(* Logix 5000 project; controller cal1632 1756-L62 rev 16.20; software revision 16.05; part 37 of 61 *)
(* tags used below, declared in another part *)
   FAULT : BOOL;
   HMI : BOOL;
   p01r09_pb_global_reset : BOOL;
   p23_ao_selected_speed : REAL;
   p23_ao_servo_ds_jog_vel_cmd : REAL;
   p23_ao_servo_ds_position_cmd : REAL;
   p23_ao_servo_ds_velocity_cmd : REAL;
   p23_ao_servo_ds_zero_offset : REAL;
   p23_ao_servo_os_jog_vel_cmd : REAL;
   p23_ao_servo_os_position_cmd : REAL;
   p23_ao_servo_os_velocity_cmd : REAL;
   p23_ao_servo_os_zero_offset : REAL;
   p23_ao_supply_selected_speed : REAL;
   p23_cpr_gear_ratio : REAL;
   p23_cpr_roll_diameter_ft : REAL;
   p23_cpr_speed_to_vfd : SYS_SPEED_TO_VFD;
   p23_di_impreg_tank_up : BOOL;
   p23_di_metering_roll : acs800_di_normal;
   p23_di_servo_ds : servo_di;
   p23_di_servo_os : servo_di;
   p23_di_supply : acs800_di_normal;
   p23_di_tank_level_high : BOOL;
   p23_di_tank_level_low : BOOL;
   p23_di_though_level_low : BOOL;
   p23_dint_to_hmi : DINT[32];
   p23_do_enable_impreg_exhaust_fan : BOOL;
   p23_do_enable_impreg_supply_fan : BOOL;
   p23_do_impreg : acs800_do_normal;
   p23_do_impreg_nip_close : BOOL;
   p23_do_servo_ds : servo_do;
   p23_do_servo_os : servo_do;
   p23_do_Spring : acs800_do_normal;
   p23_do_supply : acs800_do_normal;
   p23_servo_ds_error : SYS_ENC_WITH_ZERO_BIT;
   p23_servo_ds_warning : SYS_ENC_WITH_ZERO_BIT;
   p23_servo_os_error : SYS_ENC_WITH_ZERO_BIT;
   p23_servo_os_warning : SYS_ENC_WITH_ZERO_BIT;
   p23_spring_gear_ratio : REAL;
   p23_spring_roll_diameter_ft : REAL;
   p23_spring_speed_to_vfd : SYS_SPEED_TO_VFD;
   p23r04 : routine;
   p23r04_timer_fault : TIMER[4];
   p23r04_timer_warning : TIMER[4];
   p23r05 : routine;
   p23r05_supply_status : DINT;
   p23r05_timer_fault : TIMER[4];
   p23r05_timer_warning : TIMER[4];
   p23r11_servo_not_ready : BOOL;
   p23r11_servo_status_ab : BOOL;
   p23r11_servo_status_af : BOOL;
   p23r11_servo_status_bb : BOOL;
   p23r12_servo_not_ready : BOOL;
   p23r12_servo_status_ab : BOOL;
   p23r12_servo_status_af : BOOL;
   p23r12_servo_status_bb : BOOL;
   p23r13 : routine;
   p23r13_vfd_stopped : BOOL;
   p23r15_pid_tension_control : BOOL;
   p23r17_adjusted_speed : REAL;
   p32r13_request_auto_stop : BOOL;
(* P23_Impreg, continued *)

ROUTINE R04_Outputs   (* ladder *)
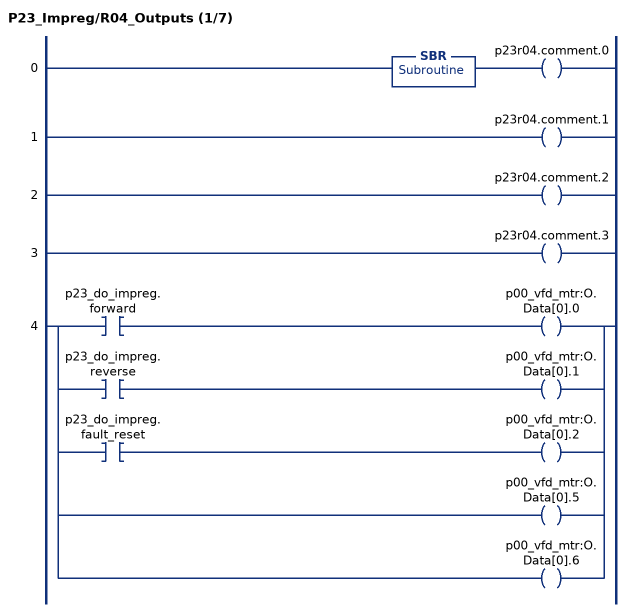
   0: SBR()OTE(p23r04.comment.0);
   1: OTE(p23r04.comment.1);
   2: OTE(p23r04.comment.2);
   3: OTE(p23r04.comment.3);
   4: [XIC(p23_do_impreg.forward) OTE(p00_vfd_mtr:O.Data[0].0) ,XIC(p23_do_impreg.reverse) OTE(p00_vfd_mtr:O.Data[0].1) ,XIC(p23_do_impreg.fault_reset) OTE(p00_vfd_mtr:O.Data[0].2) ,OTE(p00_vfd_mtr:O.Data[0].5) ,OTE(p00_vfd_mtr:O.Data[0].6) ];
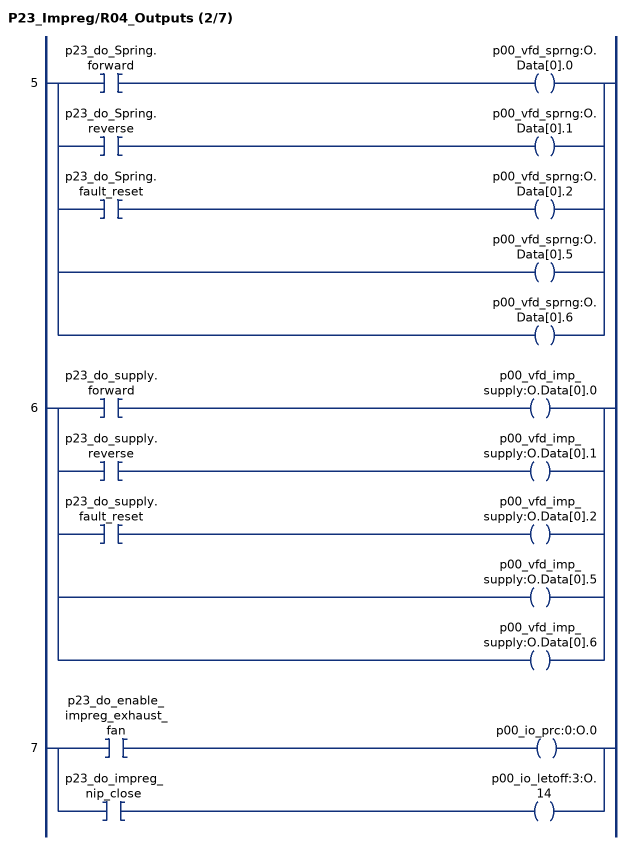
   5: [XIC(p23_do_Spring.forward) OTE(p00_vfd_sprng:O.Data[0].0) ,XIC(p23_do_Spring.reverse) OTE(p00_vfd_sprng:O.Data[0].1) ,XIC(p23_do_Spring.fault_reset) OTE(p00_vfd_sprng:O.Data[0].2) ,OTE(p00_vfd_sprng:O.Data[0].5) ,OTE(p00_vfd_sprng:O.Data[0].6) ];
   6: [XIC(p23_do_supply.forward) OTE(p00_vfd_imp_supply:O.Data[0].0) ,XIC(p23_do_supply.reverse) OTE(p00_vfd_imp_supply:O.Data[0].1) ,XIC(p23_do_supply.fault_reset) OTE(p00_vfd_imp_supply:O.Data[0].2) ,OTE(p00_vfd_imp_supply:O.Data[0].5) ,OTE(p00_vfd_imp_supply:O.Data[0].6) ];
   7: [XIC(p23_do_enable_impreg_exhaust_fan) OTE(p00_io_prc:0:O.0) ,XIC(p23_do_impreg_nip_close) OTE(p00_io_letoff:3:O.14) ];
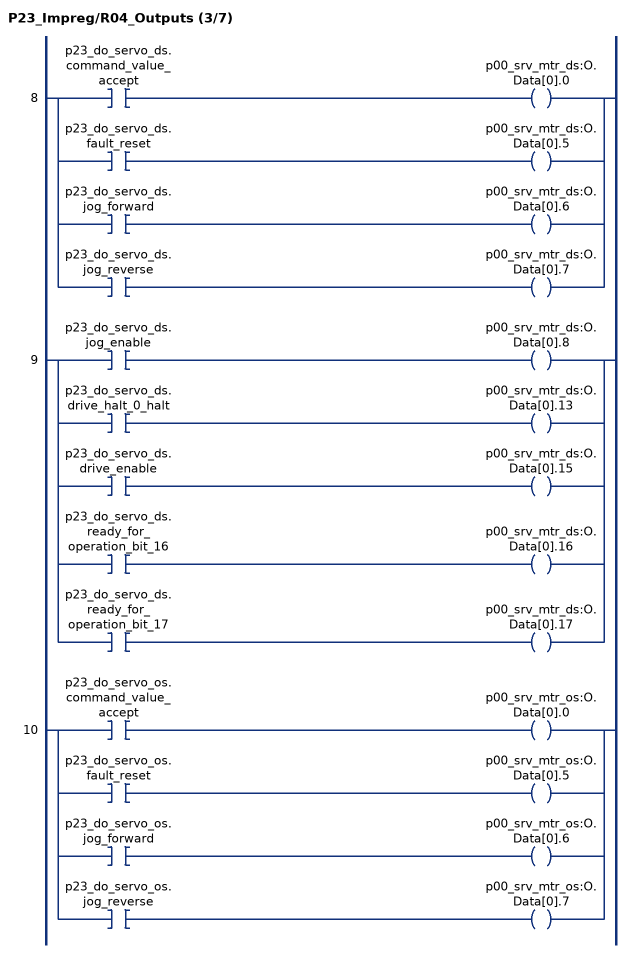
   8: [XIC(p23_do_servo_ds.command_value_accept) OTE(p00_srv_mtr_ds:O.Data[0].0) ,XIC(p23_do_servo_ds.fault_reset) OTE(p00_srv_mtr_ds:O.Data[0].5) ,XIC(p23_do_servo_ds.jog_forward) OTE(p00_srv_mtr_ds:O.Data[0].6) ,XIC(p23_do_servo_ds.jog_reverse) OTE(p00_srv_mtr_ds:O.Data[0].7) ];
   9: [XIC(p23_do_servo_ds.jog_enable) OTE(p00_srv_mtr_ds:O.Data[0].8) ,XIC(p23_do_servo_ds.drive_halt_0_halt) OTE(p00_srv_mtr_ds:O.Data[0].13) ,XIC(p23_do_servo_ds.drive_enable) OTE(p00_srv_mtr_ds:O.Data[0].15) ,XIC(p23_do_servo_ds.ready_for_operation_bit_16) OTE(p00_srv_mtr_ds:O.Data[0].16) ,XIC(p23_do_servo_ds.ready_for_operation_bit_17) OTE(p00_srv_mtr_ds:O.Data[0].17) ];
   10: [XIC(p23_do_servo_os.command_value_accept) OTE(p00_srv_mtr_os:O.Data[0].0) ,XIC(p23_do_servo_os.fault_reset) OTE(p00_srv_mtr_os:O.Data[0].5) ,XIC(p23_do_servo_os.jog_forward) OTE(p00_srv_mtr_os:O.Data[0].6) ,XIC(p23_do_servo_os.jog_reverse) OTE(p00_srv_mtr_os:O.Data[0].7) ];
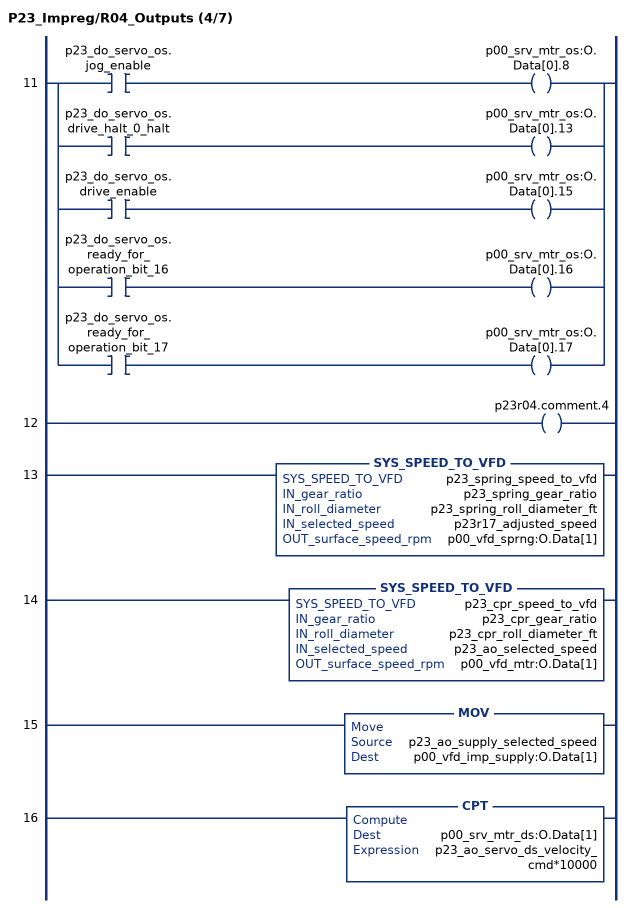
   11: [XIC(p23_do_servo_os.jog_enable) OTE(p00_srv_mtr_os:O.Data[0].8) ,XIC(p23_do_servo_os.drive_halt_0_halt) OTE(p00_srv_mtr_os:O.Data[0].13) ,XIC(p23_do_servo_os.drive_enable) OTE(p00_srv_mtr_os:O.Data[0].15) ,XIC(p23_do_servo_os.ready_for_operation_bit_16) OTE(p00_srv_mtr_os:O.Data[0].16) ,XIC(p23_do_servo_os.ready_for_operation_bit_17) OTE(p00_srv_mtr_os:O.Data[0].17) ];
   12: OTE(p23r04.comment.4);
   13: SYS_SPEED_TO_VFD(p23_spring_speed_to_vfd,p23_spring_gear_ratio,p23_spring_roll_diameter_ft,p23r17_adjusted_speed,p00_vfd_sprng:O.Data[1]);
   14: SYS_SPEED_TO_VFD(p23_cpr_speed_to_vfd,p23_cpr_gear_ratio,p23_cpr_roll_diameter_ft,p23_ao_selected_speed,p00_vfd_mtr:O.Data[1]);
   15: MOV(p23_ao_supply_selected_speed,p00_vfd_imp_supply:O.Data[1]);
   16: CPT(p00_srv_mtr_ds:O.Data[1],p23_ao_servo_ds_velocity_cmd*10000);
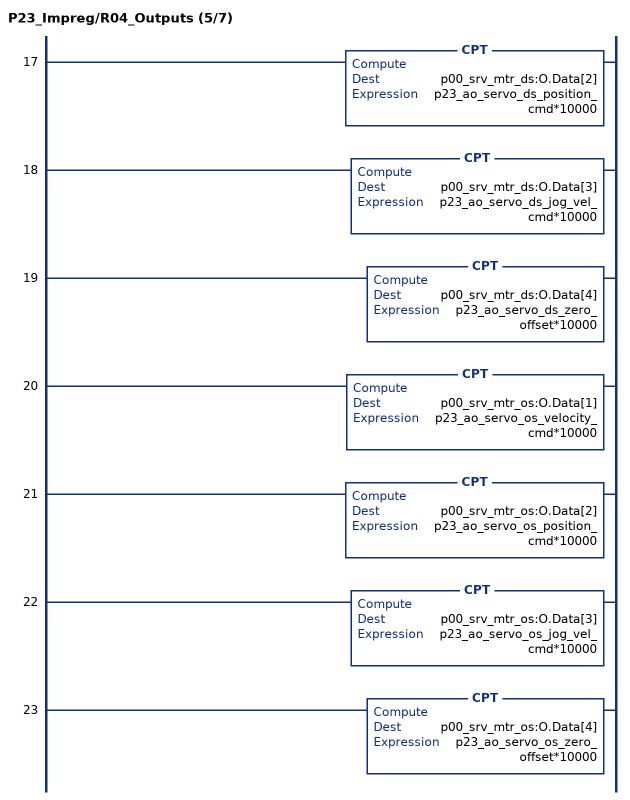
   17: CPT(p00_srv_mtr_ds:O.Data[2],p23_ao_servo_ds_position_cmd*10000);
   18: CPT(p00_srv_mtr_ds:O.Data[3],p23_ao_servo_ds_jog_vel_cmd*10000);
   19: CPT(p00_srv_mtr_ds:O.Data[4],p23_ao_servo_ds_zero_offset*10000);
   20: CPT(p00_srv_mtr_os:O.Data[1],p23_ao_servo_os_velocity_cmd*10000);
   21: CPT(p00_srv_mtr_os:O.Data[2],p23_ao_servo_os_position_cmd*10000);
   22: CPT(p00_srv_mtr_os:O.Data[3],p23_ao_servo_os_jog_vel_cmd*10000);
   23: CPT(p00_srv_mtr_os:O.Data[4],p23_ao_servo_os_zero_offset*10000);
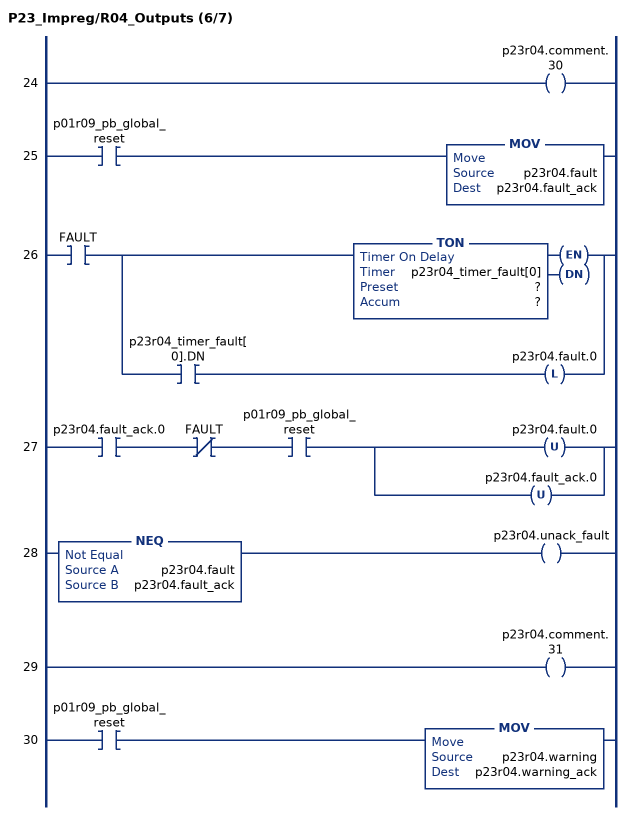
   24: OTE(p23r04.comment.30);
   25: XIC(p01r09_pb_global_reset)MOV(p23r04.fault,p23r04.fault_ack);
   26: XIC(FAULT)[TON(p23r04_timer_fault[0],?,?) ,XIC(p23r04_timer_fault[0].DN) OTL(p23r04.fault.0) ];
   27: XIC(p23r04.fault_ack.0)XIO(FAULT)XIC(p01r09_pb_global_reset)[OTU(p23r04.fault.0) ,OTU(p23r04.fault_ack.0) ];
   28: NEQ(p23r04.fault,p23r04.fault_ack)OTE(p23r04.unack_fault);
   29: OTE(p23r04.comment.31);
   30: XIC(p01r09_pb_global_reset)MOV(p23r04.warning,p23r04.warning_ack);
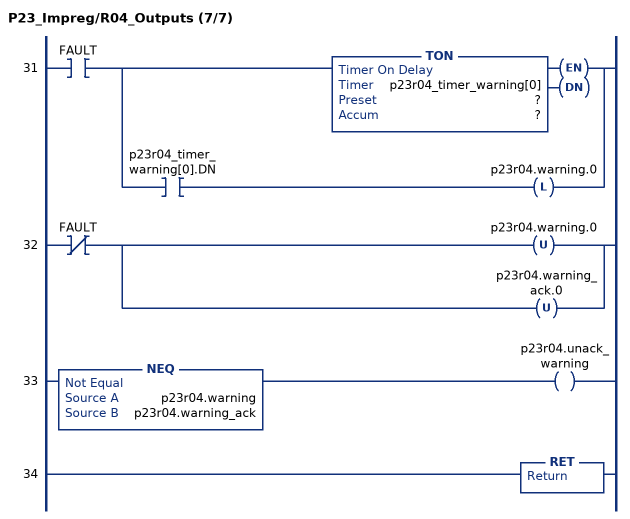
   31: XIC(FAULT)[TON(p23r04_timer_warning[0],?,?) ,XIC(p23r04_timer_warning[0].DN) OTL(p23r04.warning.0) ];
   32: XIO(FAULT)[OTU(p23r04.warning.0) ,OTU(p23r04.warning_ack.0) ];
   33: NEQ(p23r04.warning,p23r04.warning_ack)OTE(p23r04.unack_warning);
   34: RET();
END_ROUTINE

ROUTINE R05_Dint_to_HMI   (* ladder *)
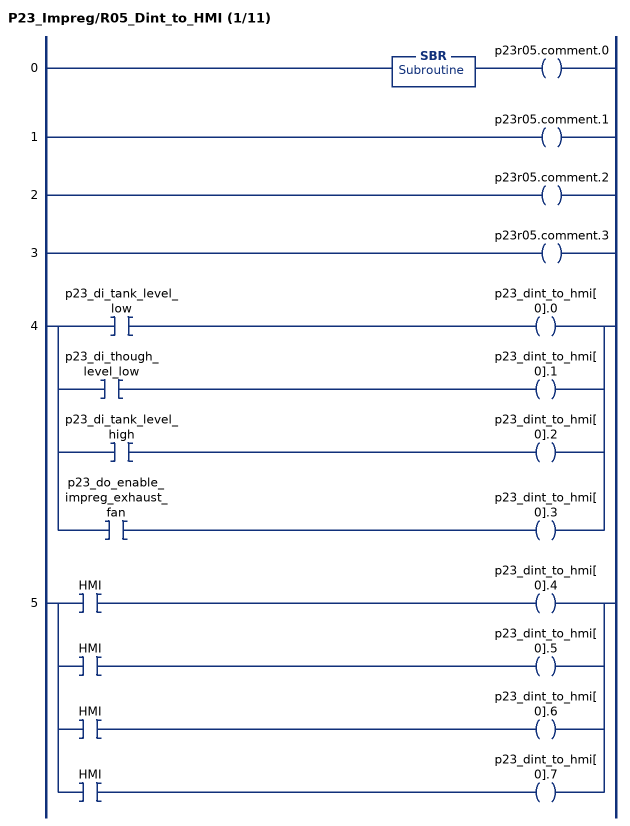
   0: SBR()OTE(p23r05.comment.0);
   1: OTE(p23r05.comment.1);
   2: OTE(p23r05.comment.2);
   3: OTE(p23r05.comment.3);
   4: [XIC(p23_di_tank_level_low) OTE(p23_dint_to_hmi[0].0) ,XIC(p23_di_though_level_low) OTE(p23_dint_to_hmi[0].1) ,XIC(p23_di_tank_level_high) OTE(p23_dint_to_hmi[0].2) ,XIC(p23_do_enable_impreg_exhaust_fan) OTE(p23_dint_to_hmi[0].3) ];
   5: [XIC(HMI) OTE(p23_dint_to_hmi[0].4) ,XIC(HMI) OTE(p23_dint_to_hmi[0].5) ,XIC(HMI) OTE(p23_dint_to_hmi[0].6) ,XIC(HMI) OTE(p23_dint_to_hmi[0].7) ];
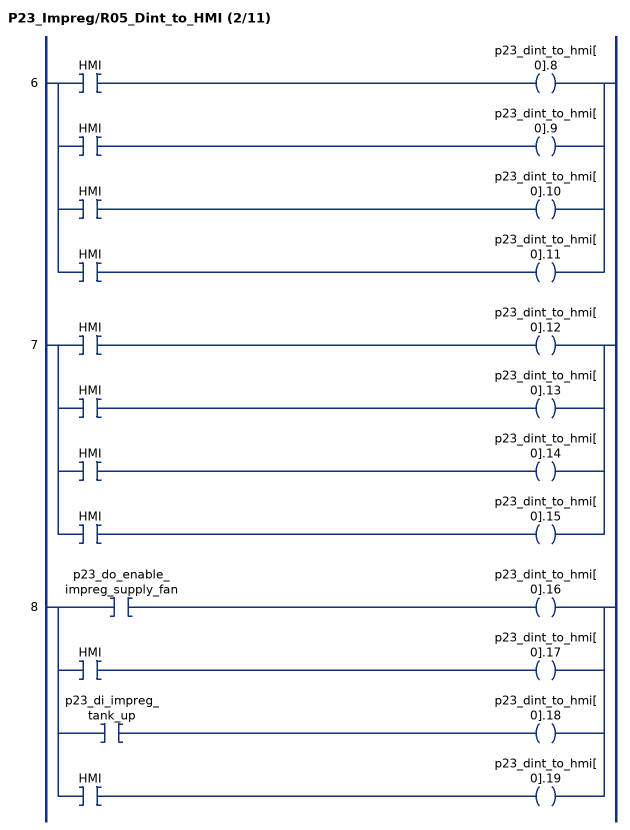
   6: [XIC(HMI) OTE(p23_dint_to_hmi[0].8) ,XIC(HMI) OTE(p23_dint_to_hmi[0].9) ,XIC(HMI) OTE(p23_dint_to_hmi[0].10) ,XIC(HMI) OTE(p23_dint_to_hmi[0].11) ];
   7: [XIC(HMI) OTE(p23_dint_to_hmi[0].12) ,XIC(HMI) OTE(p23_dint_to_hmi[0].13) ,XIC(HMI) OTE(p23_dint_to_hmi[0].14) ,XIC(HMI) OTE(p23_dint_to_hmi[0].15) ];
   8: [XIC(p23_do_enable_impreg_supply_fan) OTE(p23_dint_to_hmi[0].16) ,XIC(HMI) OTE(p23_dint_to_hmi[0].17) ,XIC(p23_di_impreg_tank_up) OTE(p23_dint_to_hmi[0].18) ,XIC(HMI) OTE(p23_dint_to_hmi[0].19) ];
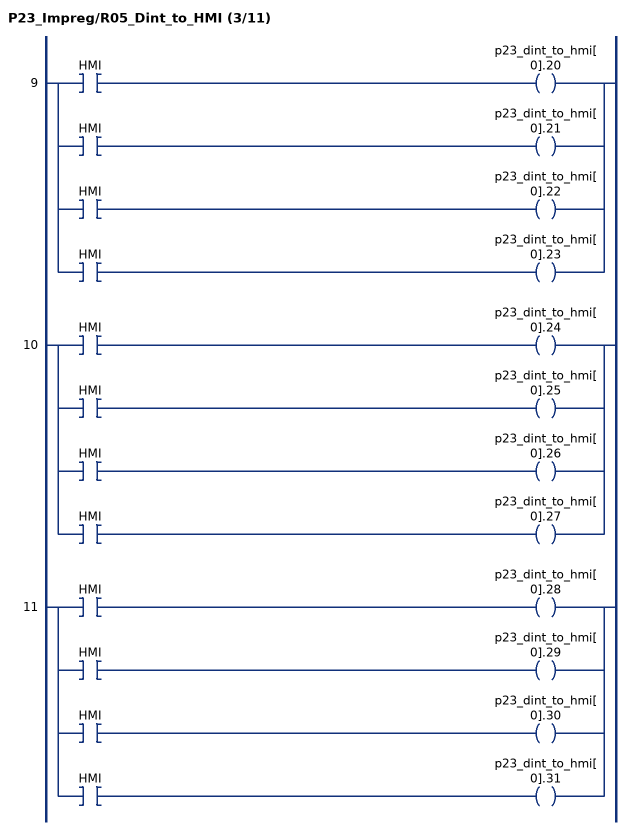
   9: [XIC(HMI) OTE(p23_dint_to_hmi[0].20) ,XIC(HMI) OTE(p23_dint_to_hmi[0].21) ,XIC(HMI) OTE(p23_dint_to_hmi[0].22) ,XIC(HMI) OTE(p23_dint_to_hmi[0].23) ];
   10: [XIC(HMI) OTE(p23_dint_to_hmi[0].24) ,XIC(HMI) OTE(p23_dint_to_hmi[0].25) ,XIC(HMI) OTE(p23_dint_to_hmi[0].26) ,XIC(HMI) OTE(p23_dint_to_hmi[0].27) ];
   11: [XIC(HMI) OTE(p23_dint_to_hmi[0].28) ,XIC(HMI) OTE(p23_dint_to_hmi[0].29) ,XIC(HMI) OTE(p23_dint_to_hmi[0].30) ,XIC(HMI) OTE(p23_dint_to_hmi[0].31) ];
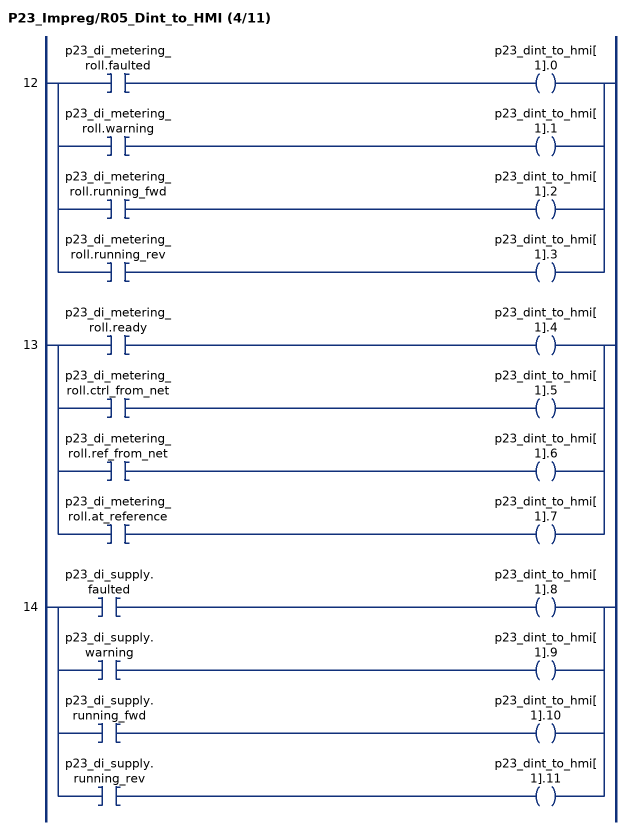
   12: [XIC(p23_di_metering_roll.faulted) OTE(p23_dint_to_hmi[1].0) ,XIC(p23_di_metering_roll.warning) OTE(p23_dint_to_hmi[1].1) ,XIC(p23_di_metering_roll.running_fwd) OTE(p23_dint_to_hmi[1].2) ,XIC(p23_di_metering_roll.running_rev) OTE(p23_dint_to_hmi[1].3) ];
   13: [XIC(p23_di_metering_roll.ready) OTE(p23_dint_to_hmi[1].4) ,XIC(p23_di_metering_roll.ctrl_from_net) OTE(p23_dint_to_hmi[1].5) ,XIC(p23_di_metering_roll.ref_from_net) OTE(p23_dint_to_hmi[1].6) ,XIC(p23_di_metering_roll.at_reference) OTE(p23_dint_to_hmi[1].7) ];
   14: [XIC(p23_di_supply.faulted) OTE(p23_dint_to_hmi[1].8) ,XIC(p23_di_supply.warning) OTE(p23_dint_to_hmi[1].9) ,XIC(p23_di_supply.running_fwd) OTE(p23_dint_to_hmi[1].10) ,XIC(p23_di_supply.running_rev) OTE(p23_dint_to_hmi[1].11) ];
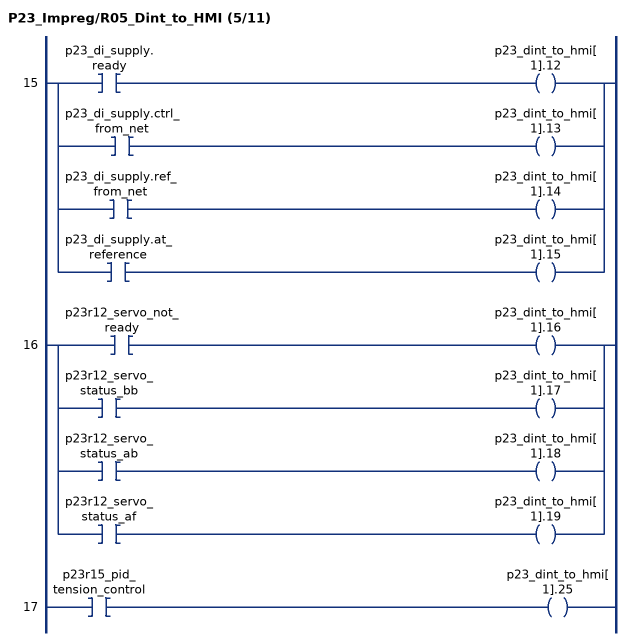
   15: [XIC(p23_di_supply.ready) OTE(p23_dint_to_hmi[1].12) ,XIC(p23_di_supply.ctrl_from_net) OTE(p23_dint_to_hmi[1].13) ,XIC(p23_di_supply.ref_from_net) OTE(p23_dint_to_hmi[1].14) ,XIC(p23_di_supply.at_reference) OTE(p23_dint_to_hmi[1].15) ];
   16: [XIC(p23r12_servo_not_ready) OTE(p23_dint_to_hmi[1].16) ,XIC(p23r12_servo_status_bb) OTE(p23_dint_to_hmi[1].17) ,XIC(p23r12_servo_status_ab) OTE(p23_dint_to_hmi[1].18) ,XIC(p23r12_servo_status_af) OTE(p23_dint_to_hmi[1].19) ];
   17: XIC(p23r15_pid_tension_control)OTE(p23_dint_to_hmi[1].25);
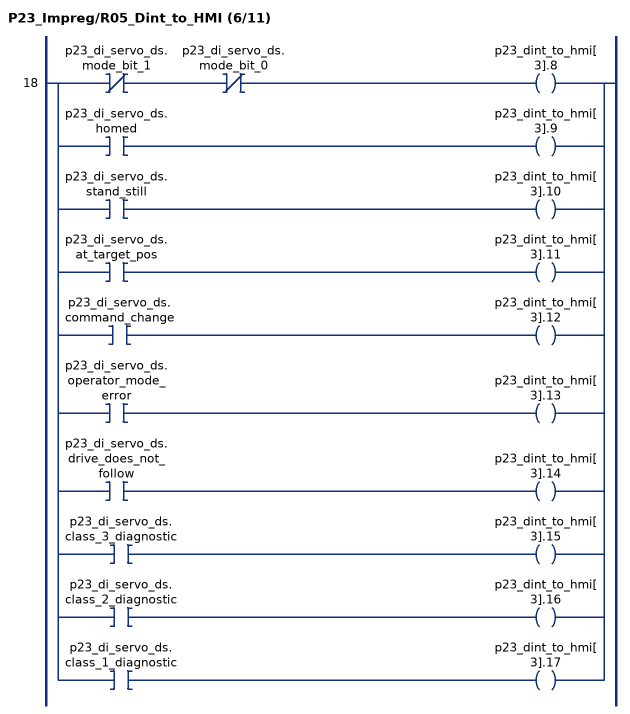
   18: [XIO(p23_di_servo_ds.mode_bit_1) XIO(p23_di_servo_ds.mode_bit_0) OTE(p23_dint_to_hmi[3].8) ,XIC(p23_di_servo_ds.homed) OTE(p23_dint_to_hmi[3].9) ,XIC(p23_di_servo_ds.stand_still) OTE(p23_dint_to_hmi[3].10) ,XIC(p23_di_servo_ds.at_target_pos) OTE(p23_dint_to_hmi[3].11) ,XIC(p23_di_servo_ds.command_change) OTE(p23_dint_to_hmi[3].12) ,XIC(p23_di_servo_ds.operator_mode_error) OTE(p23_dint_to_hmi[3].13) ,XIC(p23_di_servo_ds.drive_does_not_follow) OTE(p23_dint_to_hmi[3].14) ,XIC(p23_di_servo_ds.class_3_diagnostic) OTE(p23_dint_to_hmi[3].15) ,XIC(p23_di_servo_ds.class_2_diagnostic) OTE(p23_dint_to_hmi[3].16) ,XIC(p23_di_servo_ds.class_1_diagnostic) OTE(p23_dint_to_hmi[3].17) ];
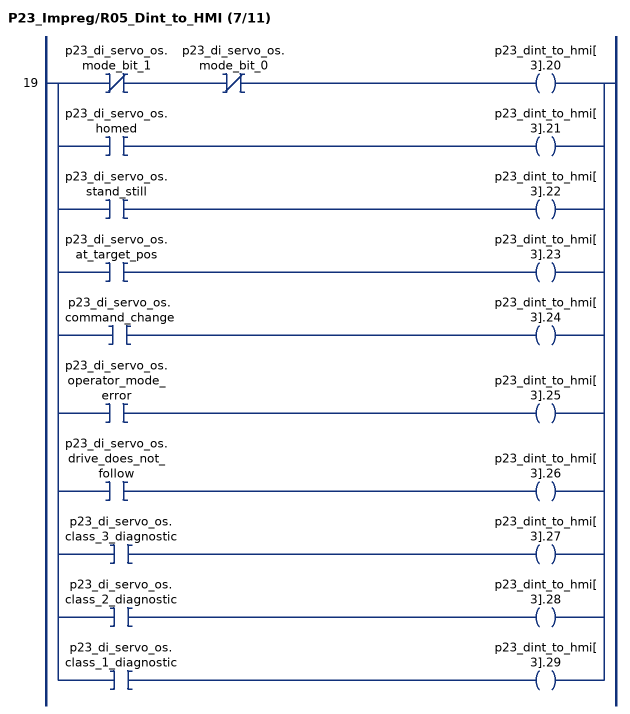
   19: [XIO(p23_di_servo_os.mode_bit_1) XIO(p23_di_servo_os.mode_bit_0) OTE(p23_dint_to_hmi[3].20) ,XIC(p23_di_servo_os.homed) OTE(p23_dint_to_hmi[3].21) ,XIC(p23_di_servo_os.stand_still) OTE(p23_dint_to_hmi[3].22) ,XIC(p23_di_servo_os.at_target_pos) OTE(p23_dint_to_hmi[3].23) ,XIC(p23_di_servo_os.command_change) OTE(p23_dint_to_hmi[3].24) ,XIC(p23_di_servo_os.operator_mode_error) OTE(p23_dint_to_hmi[3].25) ,XIC(p23_di_servo_os.drive_does_not_follow) OTE(p23_dint_to_hmi[3].26) ,XIC(p23_di_servo_os.class_3_diagnostic) OTE(p23_dint_to_hmi[3].27) ,XIC(p23_di_servo_os.class_2_diagnostic) OTE(p23_dint_to_hmi[3].28) ,XIC(p23_di_servo_os.class_1_diagnostic) OTE(p23_dint_to_hmi[3].29) ];
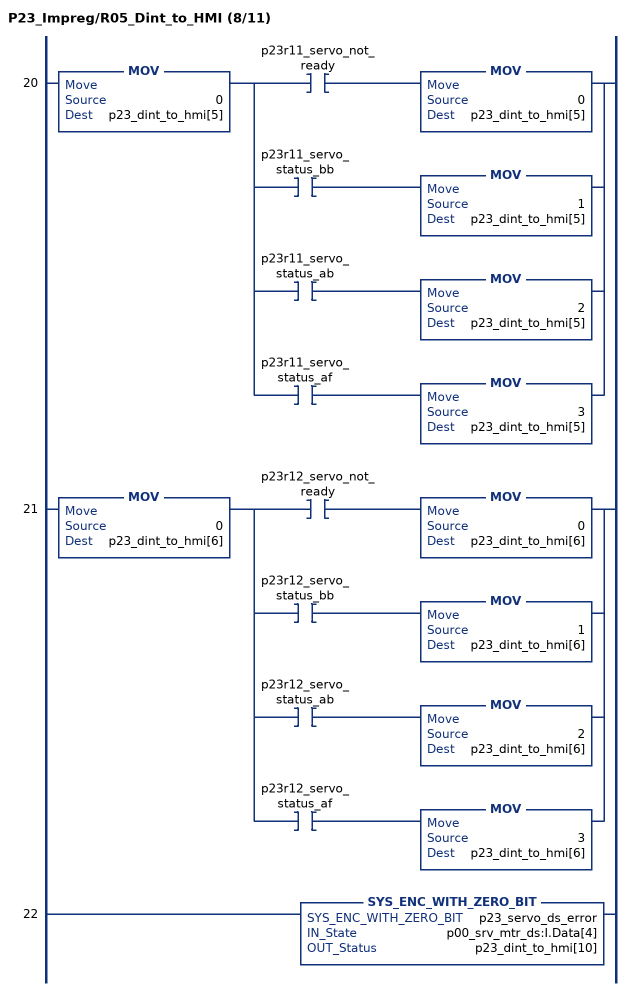
   20: MOV(0,p23_dint_to_hmi[5])[XIC(p23r11_servo_not_ready) MOV(0,p23_dint_to_hmi[5]) ,XIC(p23r11_servo_status_bb) MOV(1,p23_dint_to_hmi[5]) ,XIC(p23r11_servo_status_ab) MOV(2,p23_dint_to_hmi[5]) ,XIC(p23r11_servo_status_af) MOV(3,p23_dint_to_hmi[5]) ];
   21: MOV(0,p23_dint_to_hmi[6])[XIC(p23r12_servo_not_ready) MOV(0,p23_dint_to_hmi[6]) ,XIC(p23r12_servo_status_bb) MOV(1,p23_dint_to_hmi[6]) ,XIC(p23r12_servo_status_ab) MOV(2,p23_dint_to_hmi[6]) ,XIC(p23r12_servo_status_af) MOV(3,p23_dint_to_hmi[6]) ];
   22: SYS_ENC_WITH_ZERO_BIT(p23_servo_ds_error,p00_srv_mtr_ds:I.Data[4],p23_dint_to_hmi[10]);
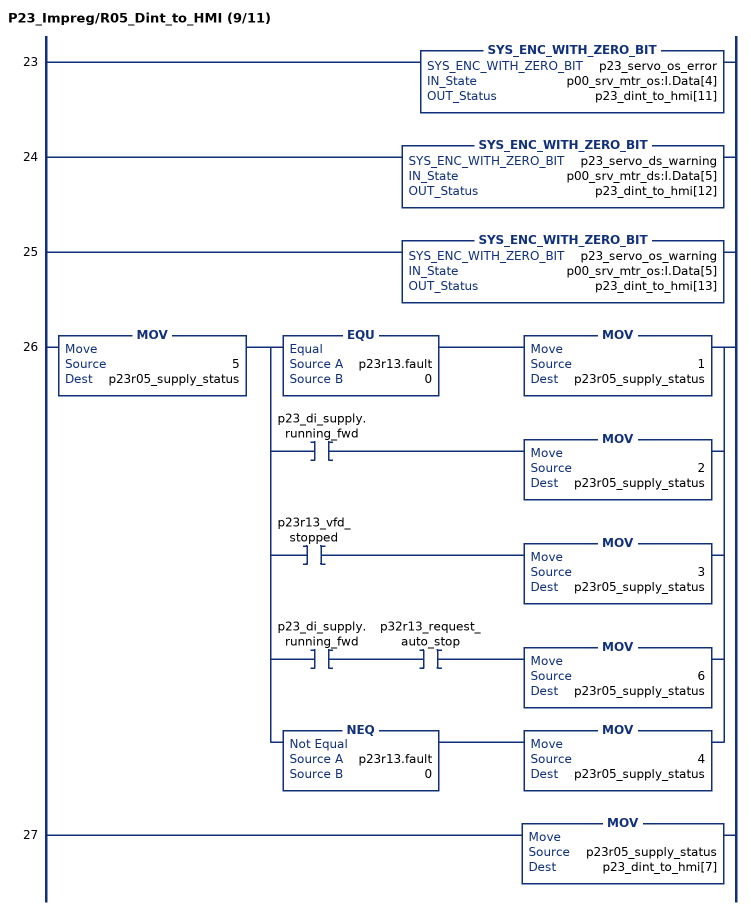
   23: SYS_ENC_WITH_ZERO_BIT(p23_servo_os_error,p00_srv_mtr_os:I.Data[4],p23_dint_to_hmi[11]);
   24: SYS_ENC_WITH_ZERO_BIT(p23_servo_ds_warning,p00_srv_mtr_ds:I.Data[5],p23_dint_to_hmi[12]);
   25: SYS_ENC_WITH_ZERO_BIT(p23_servo_os_warning,p00_srv_mtr_os:I.Data[5],p23_dint_to_hmi[13]);
   26: MOV(5,p23r05_supply_status)[EQU(p23r13.fault,0) MOV(1,p23r05_supply_status) ,XIC(p23_di_supply.running_fwd) MOV(2,p23r05_supply_status) ,XIC(p23r13_vfd_stopped) MOV(3,p23r05_supply_status) ,XIC(p23_di_supply.running_fwd) XIC(p32r13_request_auto_stop) MOV(6,p23r05_supply_status) ,NEQ(p23r13.fault,0) MOV(4,p23r05_supply_status) ];
   27: MOV(p23r05_supply_status,p23_dint_to_hmi[7]);
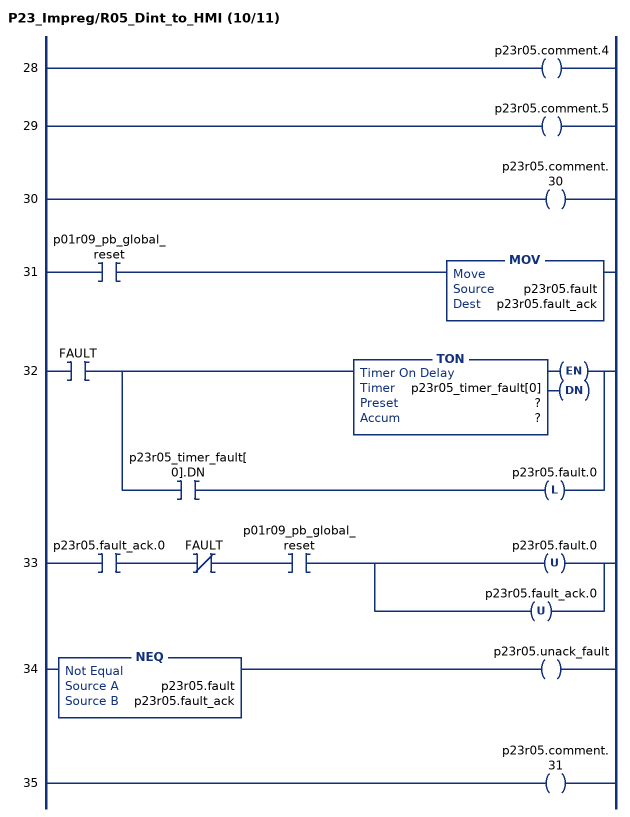
   28: OTE(p23r05.comment.4);
   29: OTE(p23r05.comment.5);
   30: OTE(p23r05.comment.30);
   31: XIC(p01r09_pb_global_reset)MOV(p23r05.fault,p23r05.fault_ack);
   32: XIC(FAULT)[TON(p23r05_timer_fault[0],?,?) ,XIC(p23r05_timer_fault[0].DN) OTL(p23r05.fault.0) ];
   33: XIC(p23r05.fault_ack.0)XIO(FAULT)XIC(p01r09_pb_global_reset)[OTU(p23r05.fault.0) ,OTU(p23r05.fault_ack.0) ];
   34: NEQ(p23r05.fault,p23r05.fault_ack)OTE(p23r05.unack_fault);
   35: OTE(p23r05.comment.31);
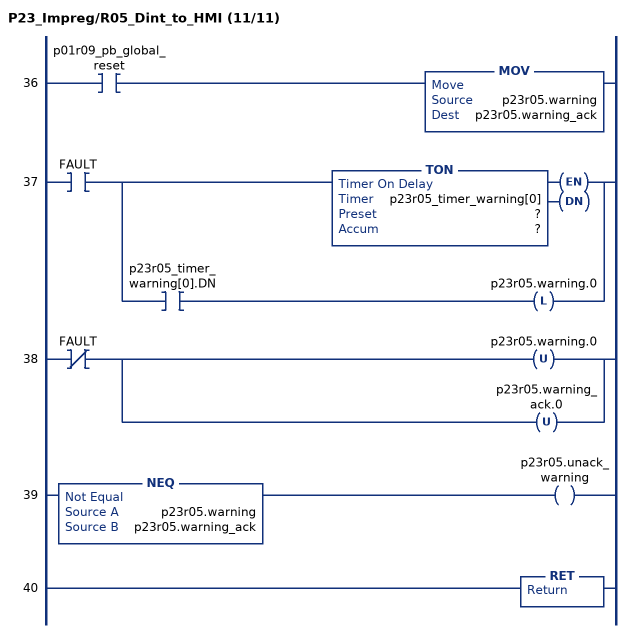
   36: XIC(p01r09_pb_global_reset)MOV(p23r05.warning,p23r05.warning_ack);
   37: XIC(FAULT)[TON(p23r05_timer_warning[0],?,?) ,XIC(p23r05_timer_warning[0].DN) OTL(p23r05.warning.0) ];
   38: XIO(FAULT)[OTU(p23r05.warning.0) ,OTU(p23r05.warning_ack.0) ];
   39: NEQ(p23r05.warning,p23r05.warning_ack)OTE(p23r05.unack_warning);
   40: RET();
END_ROUTINE
